(* Logix 5000 project; controller Sucrose_Main Emulate 5570 rev 20.12; software revision 20.01; part 26 of 30 *)
(* tags used below, declared in another part *)
   Alarm_ACK_Master_Timer : TIMER;
   ClearFault_Master : BOOL;
   DI_E23_4 : ALIAS FOR FLX_E23:4:I;   // Discrete Input EN2T_FLX 192.168.1.23
   DI_E23_5 : ALIAS FOR FLX_E23:5:I;   // Discrete Input EN2T_FLX 192.168.1.23
   DI_E25_3 : ALIAS FOR FLX_E25:3:I;   // Discrete Input EN2T_FLX 192.168.1.25
   DO_E24_0 : ALIAS FOR FLX_E24:0:O;   // Discrete Output EN2T_FLX 192.168.1.24
   DO_E24_1 : ALIAS FOR FLX_E24:1:O;   // Discrete Output EN2T_FLX 192.168.1.24
   FV230104_AOI : QSI_Flow_Valve;   // FV-23-01-04-O SUCROSE RETURN TO SUCROSE TANK #1 VALVE OPEN
   FV230204_AOI : QSI_Flow_Valve;   // FV-23-02-04-O SUCROSE RETURN TO SUCROSE TANK #2 VALVE OPEN
   FV230302_AOI : QSI_Flow_Valve;   // FV-23-03-02 SUCROSE TANK #3 INLET/SPRAYBALL VALVE
   FV230304_AOI : QSI_Flow_Valve;   // FV-23-03-04-O SUCROSE RETURN TO SUCROSE TANK #3 VALVE OPEN
   P230010_AOI : PF525_VFD_E_ENET;   // P-23-00-10 RECEIVING PUMP 1
   P230020_AOI : PF525_VFD_E_ENET;   // P-23-00-20 RECEIVING PUMP 2
   Rung_Comment : BOOL;
   Sucrose_MM_Enable : BOOL;
   SucroseCIP_RECEIVING_REMOTE : CIP_REMOTE;
   SucroseCIP_RINGMAIN_REMOTE : CIP_REMOTE;
   SucroseCIP_TK230101_REMOTE : CIP_REMOTE;
   SucroseCIP_TK230201_REMOTE : CIP_REMOTE;
   SucroseCIP_TK230301_REMOTE : CIP_REMOTE;
   SucroseDischarge : Area_Program;
   SucroseReceiving : Area_Program;
   SucroseTanks : Area_Program;
(* ReceivingArea_EN2T_IO_Discrete_DO_E25_5, continued *)

ROUTINE MainRoutine   (* ladder *)
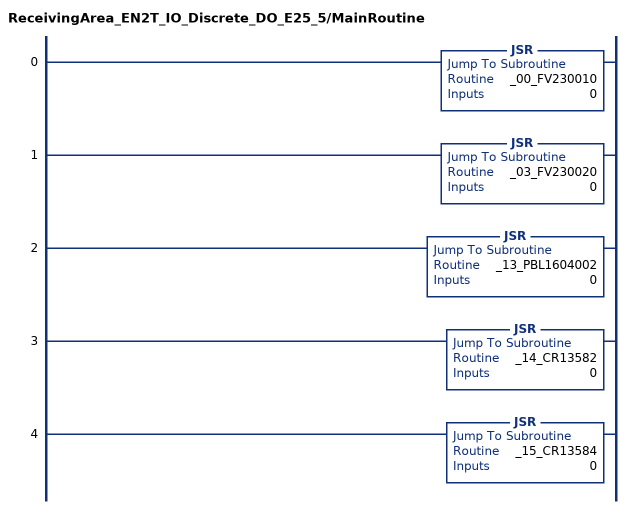
   0: JSR(_00_FV230010,0);
   1: JSR(_03_FV230020,0);
   2: JSR(_13_PBL1604002,0);
   3: JSR(_14_CR13582,0);
   4: JSR(_15_CR13584,0);
END_ROUTINE
END_PROGRAM

PROGRAM ReceivingArea_EN2T_IO_Drives   (* main routine MainRoutine *)

ROUTINE E33_P230010   (* ladder *)
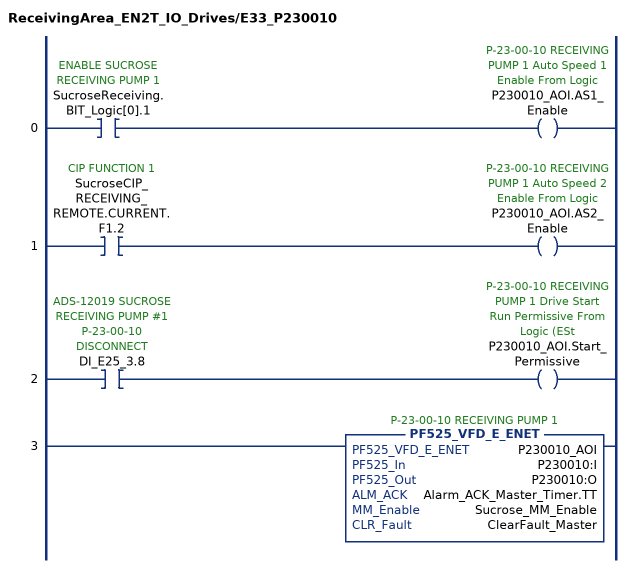
   0: XIC(SucroseReceiving.BIT_Logic[0].1)OTE(P230010_AOI.AS1_Enable);
   1: XIC(SucroseCIP_RECEIVING_REMOTE.CURRENT.F1.2)OTE(P230010_AOI.AS2_Enable);
   2: XIC(DI_E25_3.8)OTE(P230010_AOI.Start_Permissive);
   3: PF525_VFD_E_ENET(P230010_AOI,P230010:I,P230010:O,Alarm_ACK_Master_Timer.TT,Sucrose_MM_Enable,ClearFault_Master);
END_ROUTINE

ROUTINE E34_P230020   (* ladder *)
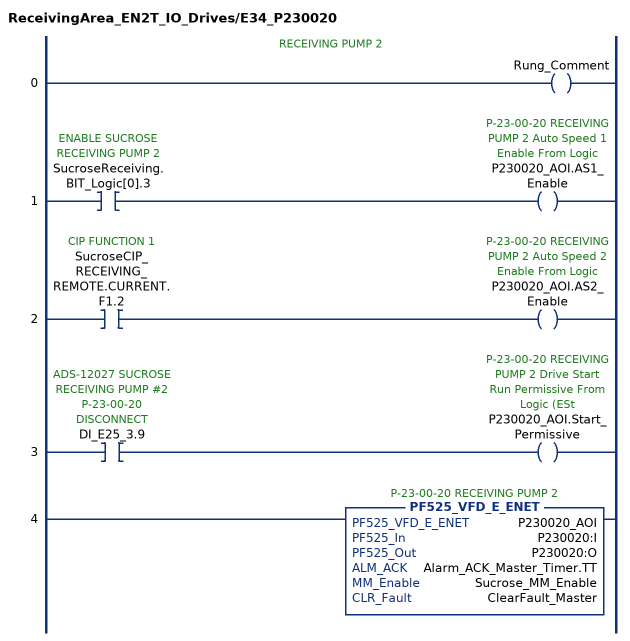
   // RECEIVING PUMP 2
   0: OTE(Rung_Comment);
   1: XIC(SucroseReceiving.BIT_Logic[0].3)OTE(P230020_AOI.AS1_Enable);
   2: XIC(SucroseCIP_RECEIVING_REMOTE.CURRENT.F1.2)OTE(P230020_AOI.AS2_Enable);
   3: XIC(DI_E25_3.9)OTE(P230020_AOI.Start_Permissive);
   4: PF525_VFD_E_ENET(P230020_AOI,P230020:I,P230020:O,Alarm_ACK_Master_Timer.TT,Sucrose_MM_Enable,ClearFault_Master);
END_ROUTINE

ROUTINE MainRoutine   (* ladder *)
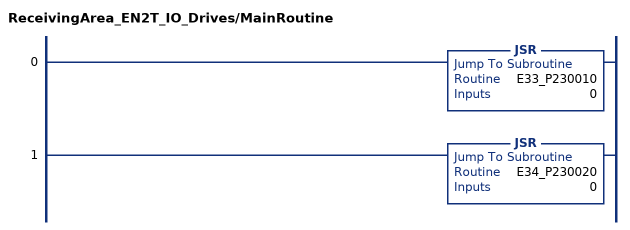
   0: JSR(E33_P230010,0);
   1: JSR(E34_P230020,0);
END_ROUTINE
END_PROGRAM

PROGRAM RecycleArea_AutoLogic   (* main routine MainRoutine *)

ROUTINE Alarm_Logic   (* ladder *)
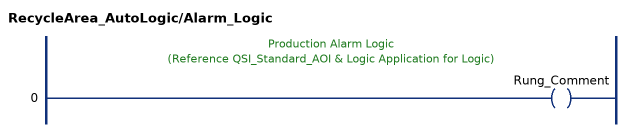
   // Production Alarm Logic
   // (Reference QSI_Standard_AOI & Logic Application for Logic)
   0: OTE(Rung_Comment);
END_ROUTINE

ROUTINE Control_Logic   (* ladder *)
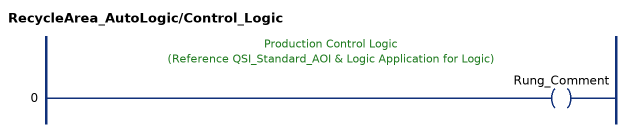
   // Production Control Logic
   // (Reference QSI_Standard_AOI & Logic Application for Logic)
   0: OTE(Rung_Comment);
END_ROUTINE

ROUTINE Enable_Logic   (* ladder *)
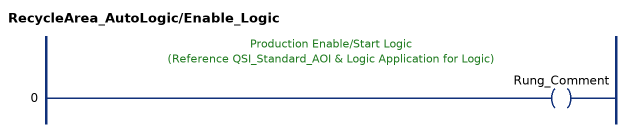
   // Production Enable/Start Logic
   // (Reference QSI_Standard_AOI & Logic Application for Logic)
   0: OTE(Rung_Comment);
END_ROUTINE

ROUTINE MainRoutine   (* ladder *)
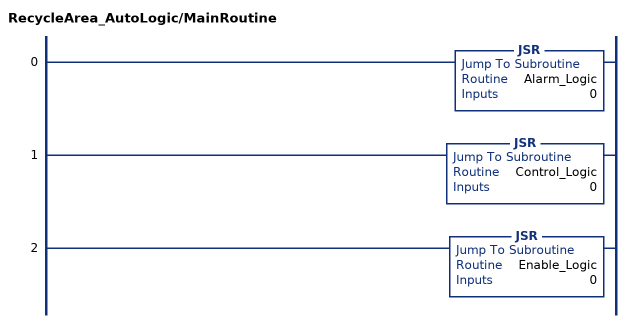
   0: JSR(Alarm_Logic,0);
   1: JSR(Control_Logic,0);
   2: JSR(Enable_Logic,0);
END_ROUTINE
END_PROGRAM

PROGRAM RecycleArea_EN2T_IO_Discrete_DO_E24_0   (* main routine MainRoutine *)

ROUTINE _05_FV230104   (* ladder *)
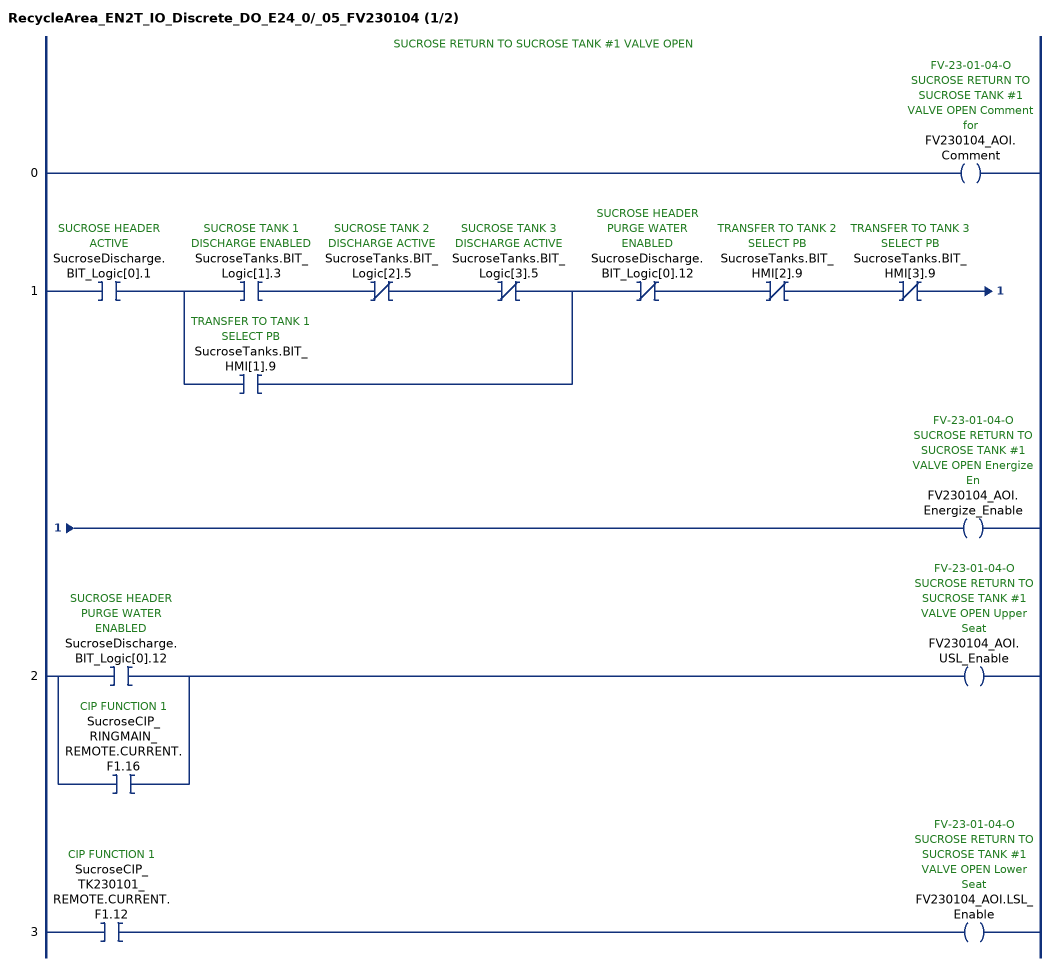
   // SUCROSE RETURN TO SUCROSE TANK #1 VALVE OPEN
   0: OTE(FV230104_AOI.Comment);
   1: XIC(SucroseDischarge.BIT_Logic[0].1)[XIC(SucroseTanks.BIT_Logic[1].3) XIO(SucroseTanks.BIT_Logic[2].5) XIO(SucroseTanks.BIT_Logic[3].5) ,XIC(SucroseTanks.BIT_HMI[1].9) ]XIO(SucroseDischarge.BIT_Logic[0].12)XIO(SucroseTanks.BIT_HMI[2].9)XIO(SucroseTanks.BIT_HMI[3].9)OTE(FV230104_AOI.Energize_Enable);
   2: [XIC(SucroseDischarge.BIT_Logic[0].12) ,XIC(SucroseCIP_RINGMAIN_REMOTE.CURRENT.F1.16) ]OTE(FV230104_AOI.USL_Enable);
   3: XIC(SucroseCIP_TK230101_REMOTE.CURRENT.F1.12)OTE(FV230104_AOI.LSL_Enable);
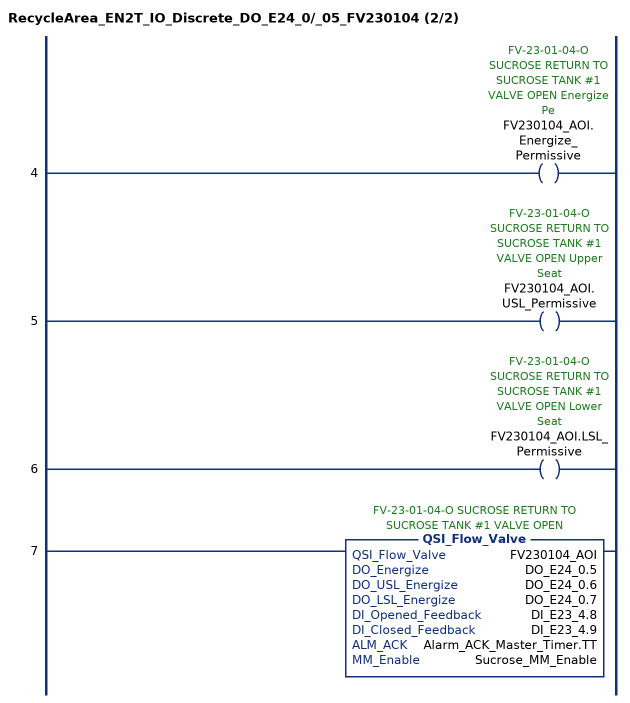
   4: OTE(FV230104_AOI.Energize_Permissive);
   5: OTE(FV230104_AOI.USL_Permissive);
   6: OTE(FV230104_AOI.LSL_Permissive);
   7: QSI_Flow_Valve(FV230104_AOI,DO_E24_0.5,DO_E24_0.6,DO_E24_0.7,DI_E23_4.8,DI_E23_4.9,Alarm_ACK_Master_Timer.TT,Sucrose_MM_Enable);
END_ROUTINE

ROUTINE _11_FV230204   (* ladder *)
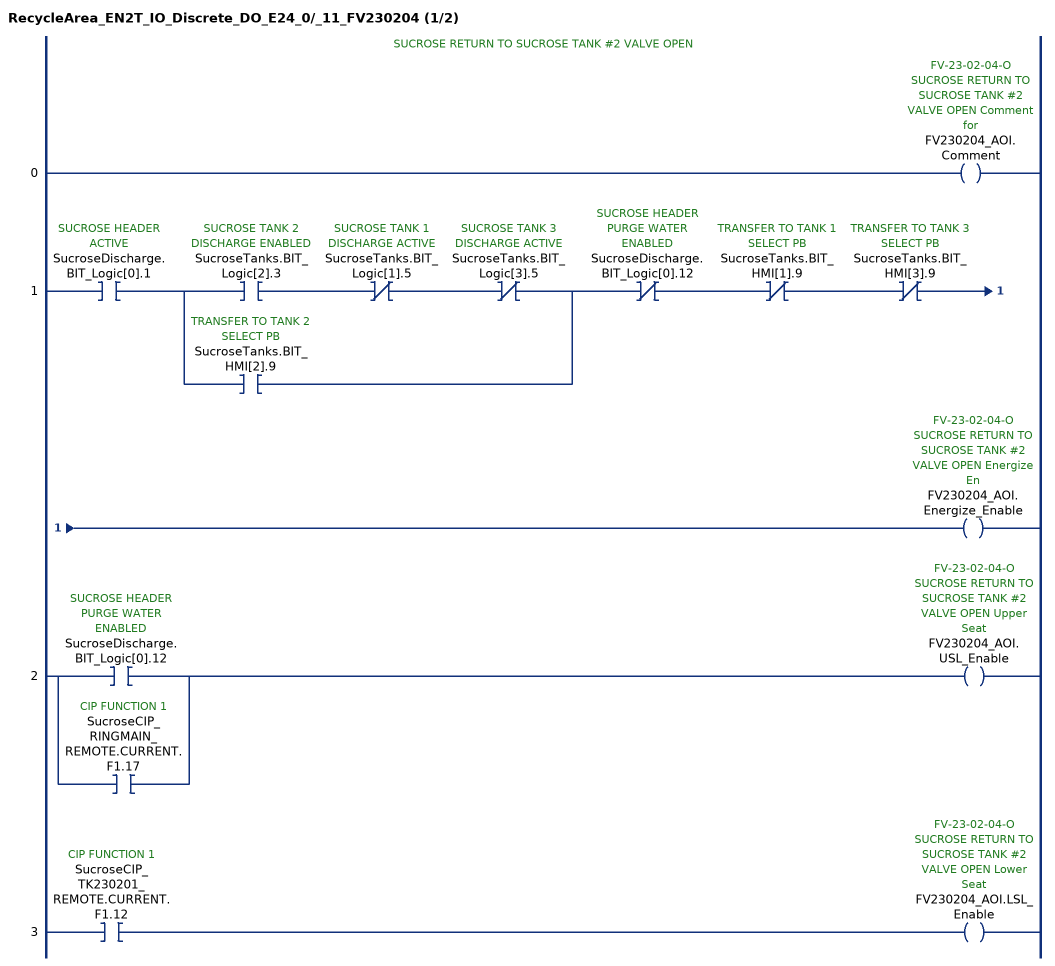
   // SUCROSE RETURN TO SUCROSE TANK #2 VALVE OPEN
   0: OTE(FV230204_AOI.Comment);
   1: XIC(SucroseDischarge.BIT_Logic[0].1)[XIC(SucroseTanks.BIT_Logic[2].3) XIO(SucroseTanks.BIT_Logic[1].5) XIO(SucroseTanks.BIT_Logic[3].5) ,XIC(SucroseTanks.BIT_HMI[2].9) ]XIO(SucroseDischarge.BIT_Logic[0].12)XIO(SucroseTanks.BIT_HMI[1].9)XIO(SucroseTanks.BIT_HMI[3].9)OTE(FV230204_AOI.Energize_Enable);
   2: [XIC(SucroseDischarge.BIT_Logic[0].12) ,XIC(SucroseCIP_RINGMAIN_REMOTE.CURRENT.F1.17) ]OTE(FV230204_AOI.USL_Enable);
   3: XIC(SucroseCIP_TK230201_REMOTE.CURRENT.F1.12)OTE(FV230204_AOI.LSL_Enable);
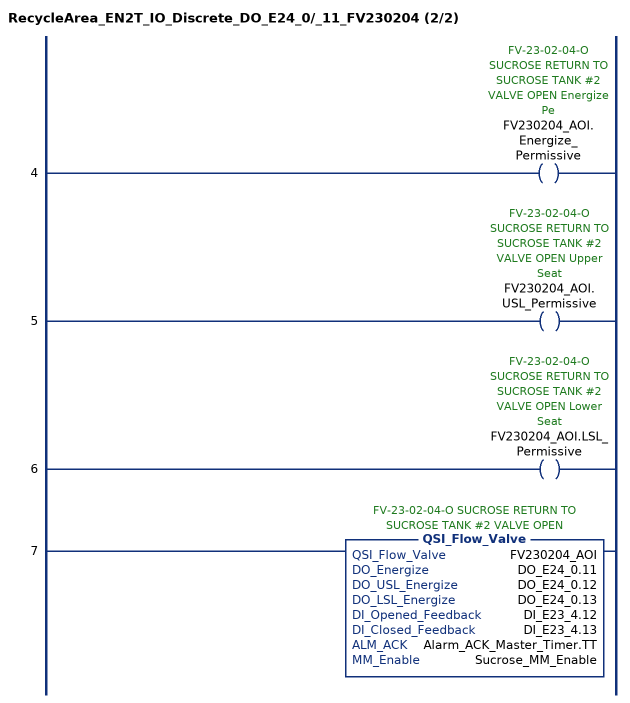
   4: OTE(FV230204_AOI.Energize_Permissive);
   5: OTE(FV230204_AOI.USL_Permissive);
   6: OTE(FV230204_AOI.LSL_Permissive);
   7: QSI_Flow_Valve(FV230204_AOI,DO_E24_0.11,DO_E24_0.12,DO_E24_0.13,DI_E23_4.12,DI_E23_4.13,Alarm_ACK_Master_Timer.TT,Sucrose_MM_Enable);
END_ROUTINE

ROUTINE MainRoutine   (* ladder *)
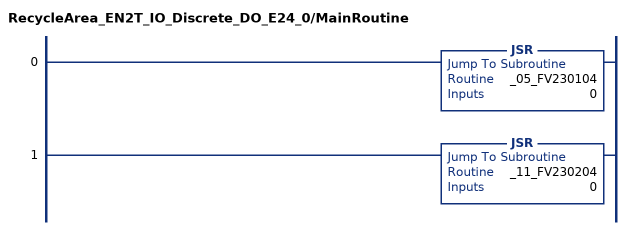
   0: JSR(_05_FV230104,0);
   1: JSR(_11_FV230204,0);
END_ROUTINE
END_PROGRAM

PROGRAM RecycleArea_EN2T_IO_Discrete_DO_E24_1   (* main routine MainRoutine *)

ROUTINE _03_FV230304   (* ladder *)
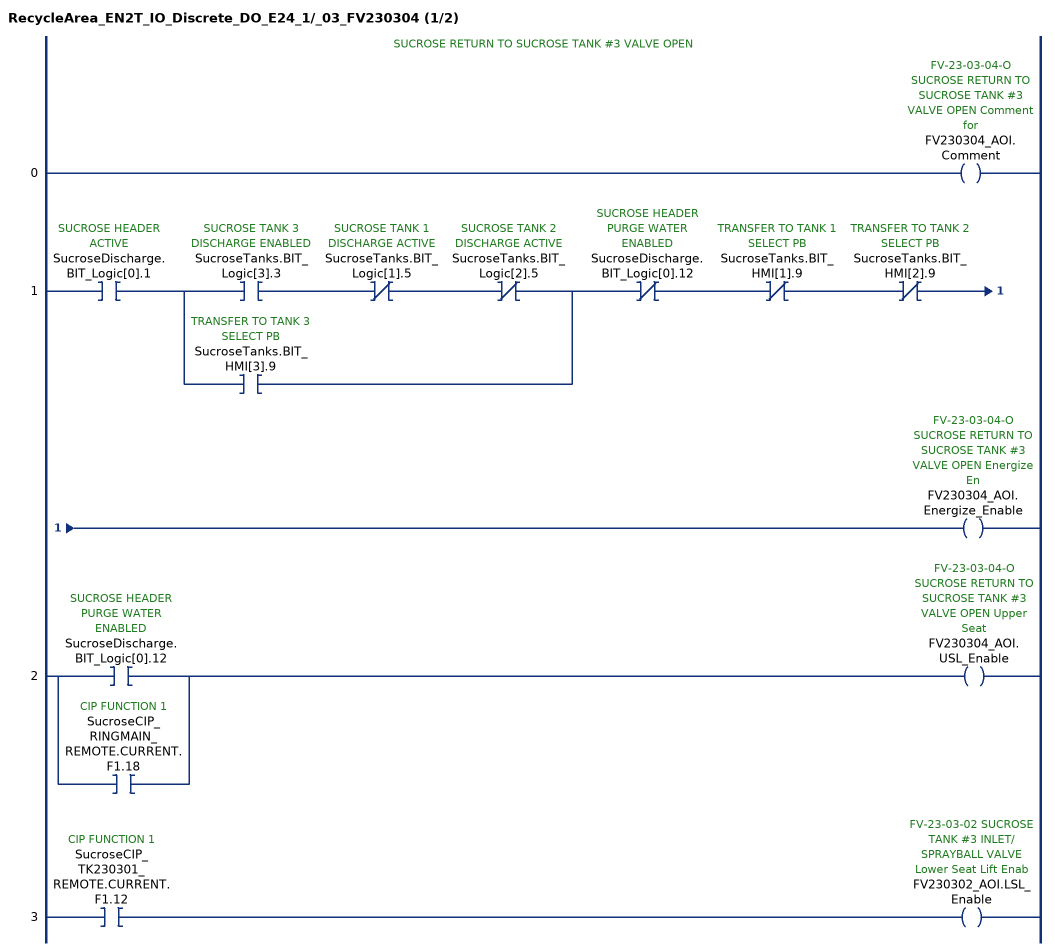
   // SUCROSE RETURN TO SUCROSE TANK #3 VALVE OPEN
   0: OTE(FV230304_AOI.Comment);
   1: XIC(SucroseDischarge.BIT_Logic[0].1)[XIC(SucroseTanks.BIT_Logic[3].3) XIO(SucroseTanks.BIT_Logic[1].5) XIO(SucroseTanks.BIT_Logic[2].5) ,XIC(SucroseTanks.BIT_HMI[3].9) ]XIO(SucroseDischarge.BIT_Logic[0].12)XIO(SucroseTanks.BIT_HMI[1].9)XIO(SucroseTanks.BIT_HMI[2].9)OTE(FV230304_AOI.Energize_Enable);
   2: [XIC(SucroseDischarge.BIT_Logic[0].12) ,XIC(SucroseCIP_RINGMAIN_REMOTE.CURRENT.F1.18) ]OTE(FV230304_AOI.USL_Enable);
   3: XIC(SucroseCIP_TK230301_REMOTE.CURRENT.F1.12)OTE(FV230302_AOI.LSL_Enable);
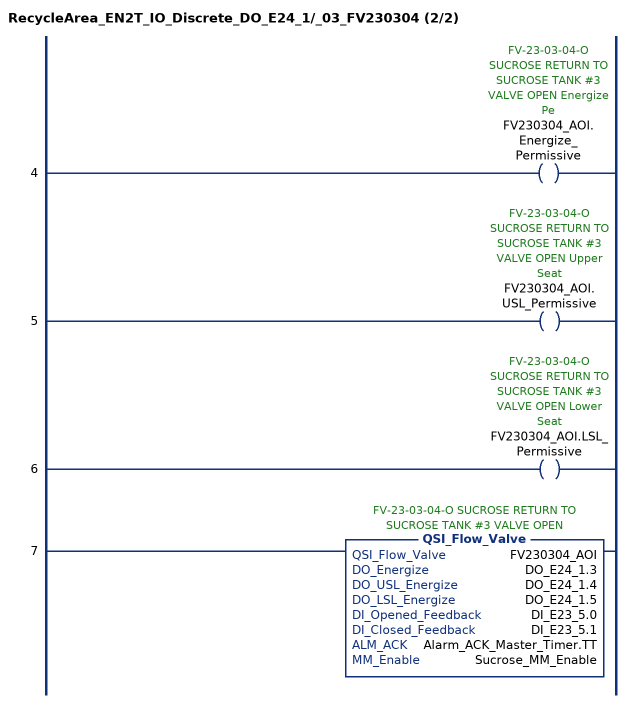
   4: OTE(FV230304_AOI.Energize_Permissive);
   5: OTE(FV230304_AOI.USL_Permissive);
   6: OTE(FV230304_AOI.LSL_Permissive);
   7: QSI_Flow_Valve(FV230304_AOI,DO_E24_1.3,DO_E24_1.4,DO_E24_1.5,DI_E23_5.0,DI_E23_5.1,Alarm_ACK_Master_Timer.TT,Sucrose_MM_Enable);
END_ROUTINE

ROUTINE MainRoutine   (* ladder *)
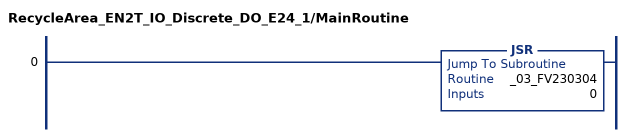
   0: JSR(_03_FV230304,0);
END_ROUTINE
END_PROGRAM

PROGRAM Steam_AirArea_AutoLogic   (* main routine MainRoutine *)

ROUTINE Alarm_Logic   (* ladder *)
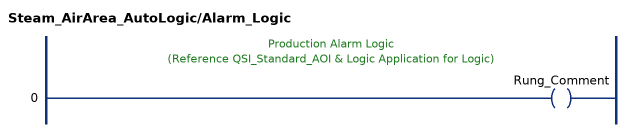
   // Production Alarm Logic
   // (Reference QSI_Standard_AOI & Logic Application for Logic)
   0: OTE(Rung_Comment);
END_ROUTINE

ROUTINE Control_Logic   (* ladder *)
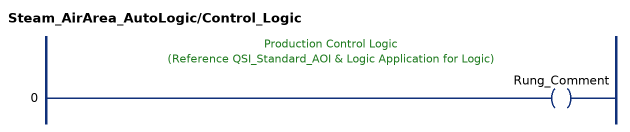
   // Production Control Logic
   // (Reference QSI_Standard_AOI & Logic Application for Logic)
   0: OTE(Rung_Comment);
END_ROUTINE
